// Mitsubishi GX Works2 project: LATCH   PLC: Q03UDV

PROGRAM MAIN
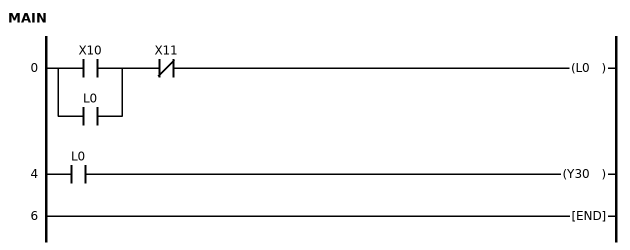
0     LD      X10
      OR      L0
      ANI     X11
      OUT     L0
4     LD      L0
      OUT     Y30
6     END
END_PROGRAM
